FUNCTION_BLOCK SENSOR_ADCPI
  {SET_ATTRIBUTE(OpcUa, DEVICE.SENSOR)}
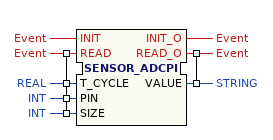
  EVENT_INPUT
    INIT;
    READ WITH T_CYCLE, PIN, SIZE;
  END_EVENT
  EVENT_OUTPUT
    INIT_O;
    READ_O WITH VALUE;
  END_EVENT
  VAR_INPUT
    T_CYCLE : REAL; {SET_ATTRIBUTE(OpcUa, Variable)}
    PIN : INT; {SET_ATTRIBUTE(OpcUa, Variable)}
    SIZE : INT; {SET_ATTRIBUTE(OpcUa, Variable)}
  END_VAR
  VAR_OUTPUT
    VALUE : STRING; {SET_ATTRIBUTE(OpcUa, Variable)}
  END_VAR
END_FUNCTION_BLOCK
